{attribute 'GeneratedUsingTerminal: ELX9560-0000-0018'}
{attribute addProperty BoxType "ELX9560-0000-0018"}
{attribute addProperty Id "EtcSlaveTerminalBaseStatus_UinAT %I*Status_Uin_627CC56E1Status_UexAT %I*Status_Uex_834F30501WcStateAT %I*WcState_9091E0EB2InfoDataAT %I*InfoData_6F19DB2B2"}
{attribute addProperty CRC "3227245878"}
{attribute addProperty Size "6"}
TYPE ELX9560_C05BDD36 EXTENDS EtcSlaveTerminalBase :
STRUCT
	{attribute addProperty Name "Status_Uin"}
	Status_Uin : Status_Uin_627CC56E;
	{attribute addProperty Name "Status_Uex"}
	Status_Uex : Status_Uex_834F3050;
	{attribute addProperty Name "WcState"}
	WcState : WcState_9091E0EB;
	{attribute addProperty Name "InfoData"}
	InfoData : InfoData_6F19DB2B;
END_STRUCT
END_TYPE

(* stored: Version 1.2.0.0, ProductVersion 3.1.4024.9
   DUT ELX9560_C05BDD36: Id {fffeb33f-9202-4cac-956b-6c92440326e9} *)
